// TIA Portal V18 export
TYPE "KukaRobot_SysInput"
   STRUCT
      SI : Struct
         PGNO_PBIT : Byte;
         PGNO_PARITY : Bool;
         PGNO_VALID : Bool;
         EXT_START : Bool;
         MOVE_ENABLE : Bool;
         CONF_MESS : Bool;
         DRIVES_OFF : Bool;
         DRIVES_ON : Bool;
         I_O_ACT : Bool;
         di_17 : Bool;
         di_18 : Bool;
         di_19 : Bool;
         di_20 : Bool;
         di_21 : Bool;
         di_22 { ExternalVisible := 'False'} : Bool;
         di_23 : Bool;
         di_24 : Bool;
         di_25 : Bool;
         di_26 : Bool;
         di_27 : Bool;
         di_28 : Bool;
         di_29 : Bool;
         di_30 : Bool;
         di_31 : Bool;
         di_32 : Bool;
         di_33 : Bool;
         di_34 : Bool;
         di_35 : Bool;
         di_36 : Bool;
         di_37 : Bool;
         di_38 : Bool;
         di_39 : Bool;
         di_40 : Bool;
         di_41 : Bool;
         di_42 : Bool;
         di_43 : Bool;
         di_44 : Bool;
         di_45 : Bool;
         di_46 : Bool;
         di_47 : Bool;
         di_48 : Bool;
      END_STRUCT;
   END_STRUCT;
END_TYPE
